(* IEC 61131-3 sources: Std_PalletMover/Class/Dana_Tm4, 1 file *)

(* ---- Dana_Tm4.st ---- *)
(*!
<Class
	Name               = "Dana_Tm4"
	Revision           = "0.0"
	RealtimeTask       = "false"
	CyclicTask         = "true"
	BackgroundTask     = "false"
	Sigmatek           = "false"
	OSInterface        = "false"
	HighPriority       = "false"
	Automatic          = "false"
	UpdateMode         = "Prescan"
	SharedCommandTable = "true"
	Objectsize         = "(900,180)">
	<Channels>
		<Server Name="ActualEncoder" Visualized="false" Initialize="false" WriteProtected="true" Retentive="false"/>
		<Server Name="ActualSpeed" Visualized="false" Initialize="false" WriteProtected="true" Retentive="false"/>
		<Server Name="ActualTorque" Visualized="false" Initialize="false" WriteProtected="true" Retentive="false"/>
		<Server Name="BatteryLevel" Visualized="false" Initialize="false" WriteProtected="true" Retentive="false"/>
		<Server Name="BatteryVoltage" Visualized="false" Initialize="false" WriteProtected="true" Retentive="false"/>
		<Server Name="InverterTemp" Visualized="false" Initialize="false" WriteProtected="true" Retentive="false"/>
		<Server Name="MotorControl" Visualized="false" Initialize="false" WriteProtected="true" Retentive="false"/>
		<Server Name="MotorError" Visualized="false" Initialize="false" WriteProtected="true" Retentive="false"/>
		<Server Name="MotorLoad" Visualized="false" Initialize="false" WriteProtected="true" Retentive="false"/>
		<Server Name="MotorState" Visualized="false" Initialize="false" WriteProtected="false" Retentive="false"/>
		<Server Name="MotorTemp" Visualized="false" Initialize="false" WriteProtected="true" Retentive="false"/>
		<Server Name="SetFeedForward" Visualized="false" Initialize="false" WriteProtected="true" Retentive="false"/>
		<Server Name="SetSpeed" Visualized="false" Initialize="false" WriteProtected="true" Retentive="false"/>
	</Channels>
	<Network Name="Dana_Tm4">
		<!-- List of Components in this network -->
		<Components>
			<Object
				Name       = "_base"
				Class      = "CanOpenWewoBase"
				Position   = "(218,120)"
				Visualized = "false">
				<Channels>
					<Server Name="Server0"/>
					<Client Name="cNode"/>
					<Client Name="ConfigData"/>
					<Client Name="Driver"/>
				</Channels>
			</Object>
		</Components>
		<Comments>
		</Comments>
		<!-- List of Connections in this network -->
		<Connections>
			<Connection Source="this.Server0" Destination="_base.Server0" Vertices="(946,210),(774,210),"/>
			<Connection Source="_base.cNode" Destination="this.cNode" Vertices="(218,270),(38,270),"/>
			<Connection Source="_base.Driver" Destination="this.Driver" Vertices="(218,210),(38,210),"/>
		</Connections>
		<!-- Headerfiles -->
		<Options>
		</Options>
	</Network>
</Class>
*)
#pragma using CanOpenWewoBase

Dana_Tm4 : CLASS
: CanOpenWewoBase
	TYPE
	  tControlWord : BINT  //! <Type Public="true" Name="tControlWord"/>
	  [
	    1 DriveEnable,
	    2 MainContactor,
	    3 BrakeRelease,
	    4 Output_01,
	    5 Output_02,
	    6 Output_03,
	    7 Output_04,
	    8 SafeStop,
	    9 Bit9,
	    10 Bit10,
	    11 Bit11,
	    12 Bit12,
	    13 Bit13,
	    14 Bit14,
	    15 Bit15,
	    16 Reset,
	  ];
#pragma pack(push, 1)
	  tCurrent : STRUCT
	    StructItem : SINT;
	    StructItem0 : SINT;
	  END_STRUCT;
#pragma pack(pop)
	  tStatusbyte : BSINT  //! <Type Public="true" Name="tStatusbyte"/>
	  [
	    1 PowerActive,
	    2 Fault,
	    3 TorqueMode,
	    4 ModeAnalog,
	    5 ModeCan,
	    6 ccwActive,
	    7 SafeStopActive,
	    8 ToggelBit,
	  ];
	END_TYPE
  //Servers:
	MotorState 	: SvrCh_gt_AgvMotorState;
	MotorLoad 	: SvrCh_DINT;
	ActualSpeed 	: SvrCh_DINT;
	ActualTorque 	: SvrCh_DINT;
	ActualEncoder 	: SvrCh_DINT;
	MotorError 	: SvrCh_DINT;
	BatteryLevel 	: SvrCh_DINT;
	InverterTemp 	: SvrCh_DINT;
	MotorTemp 	: SvrCh_DINT;
	BatteryVoltage 	: SvrCh_DINT;
	SetSpeed 	: SvrCh_DINT;
	SetFeedForward 	: SvrCh_DINT;
	MotorControl 	: SvrCh_gt_AgvMotorControl;
  //Clients:
  //Variables:
		MotorStatus 	: tStatusbyte;
		MotorCntr 	: tControlWord;
		Current 	: tCurrent;
		CurrendState 	: gt_AgvMotorState;
		ReqState 	: gt_AgvMotorState;
		LastToggelBit 	: DINT;
		LasttAlive 	: UDINT;
		MotorTimeOut 	: DINT;
  //Functions:

	FUNCTION VIRTUAL GLOBAL CyWork
		VAR_INPUT
			EAX 	: UDINT;
		END_VAR
		VAR_OUTPUT
			state (EAX) 	: UDINT := READY;
		END_VAR;

	FUNCTION GetdataCan;

	FUNCTION SetdataCan;

	FUNCTION GLOBAL Method;

	FUNCTION HandelStates;

	FUNCTION CheckError;

	FUNCTION VIRTUAL GLOBAL MotorState::Read
		VAR_OUTPUT
			output (EAX) 	: gt_AgvMotorState;
		END_VAR;

	FUNCTION VIRTUAL GLOBAL MotorState::Write
		VAR_INPUT
			input (EAX) 	: gt_AgvMotorState;
		END_VAR
		VAR_OUTPUT
			result (EAX) 	: gt_AgvMotorState;
		END_VAR;
  //Tables:
	FUNCTION @STD
		VAR_OUTPUT
			ret_code	: CONFSTATES;
		END_VAR;
	FUNCTION GLOBAL TAB @CT_;
END_CLASS;

FUNCTION VIRTUAL GLOBAL Dana_Tm4::CyWork
	VAR_INPUT
		EAX 	: UDINT;
	END_VAR
	VAR_OUTPUT
		state (EAX) 	: UDINT;(* := READY *)
	END_VAR

     GetdataCan();

     HandelStates();

     SetDataCan();

END_FUNCTION

FUNCTION Dana_Tm4::GetdataCan

    VAR
    	Pdata : ^CanObjStr;
    END_VAR

     Pdata := GetPDO(PdoId:=16#180);
    if Pdata <> nil then
         MotorStatus    := Pdata^.Data[1];
         MotorLoad      := Pdata^.Data[2];
         ActualTorque   := Pdata^.Data[3]$int;
         ActualSpeed    := Pdata^.Data[5]$int;
         ActualEncoder := Pdata^.Data[7]$int;
    END_IF;

    Pdata := GetPDO(PdoId:=16#280);
    if Pdata <> nil then
        MotorError      := Pdata^.Data[1]$int;
        BatteryLevel     :=Pdata^.Data[3];
        InverterTemp    :=Pdata^.Data[4];
        MotorTemp       :=Pdata^.Data[5]$int;
        BatteryVoltage  :=Pdata^.Data[7]$int;
    end_if;

END_FUNCTION

FUNCTION Dana_Tm4::SetdataCan

SendPDO(PdoId:=16#200, Bytes:=8, Value1:=MotorCntr$INT, Value2:=SetSpeed$int, Value3:=SetFeedForward$int, Value4:=Current$int);

END_FUNCTION

FUNCTION VIRTUAL GLOBAL Dana_Tm4::MotorState::Write
	VAR_INPUT
		input (EAX) 	: gt_AgvMotorState;
	END_VAR
	VAR_OUTPUT
		result (EAX) 	: gt_AgvMotorState;
	END_VAR

	MotorState := ::gt_AgvMotorState::M_St_Busy;;
    ReqState := input;
	result := ::gt_AgvMotorState::M_St_Busy;

END_FUNCTION

FUNCTION GLOBAL Dana_Tm4::Method

END_FUNCTION

FUNCTION Dana_Tm4::HandelStates

    case CurrendState of

        ::gt_AgvMotorState::M_St_Config:

        ::gt_AgvMotorState::M_St_Error:

        ::gt_AgvMotorState::M_St_Ready:
            CheckError();
            MotorState := ::gt_AgvMotorState::M_St_Ready;

        ::gt_AgvMotorState::M_St_Operational:
               CheckError();

        ::gt_AgvMotorState::M_St_Reset:
             if LastToggelBit <> MotorStatus.ToggelBit then
                CurrendState :=  ::gt_AgvMotorState::M_St_Ready;
                MotorState := ::gt_AgvMotorState::M_St_Ready;
            end_if;

    end_case;

    case ReqState of

          ::gt_AgvMotorState::M_St_Reset:
            MotorCntr.Reset := true;
            CurrendState :=  ::gt_AgvMotorState::M_St_Reset;
            ReqState := ::gt_AgvMotorState::M_St_Busy;
            LastToggelBit := MotorStatus.ToggelBit;

           ::gt_AgvMotorState::M_St_Busy:

    end_case;

END_FUNCTION

FUNCTION VIRTUAL GLOBAL Dana_Tm4::MotorState::Read
	VAR_OUTPUT
		output (EAX) 	: gt_AgvMotorState;
	END_VAR

    MotorState := CurrendState;
	output := MotorState;

END_FUNCTION

FUNCTION Dana_Tm4::CheckError
    if tAlive = LasttAlive then
        MotorTimeOut -=1;
        if MotorTimeOut <= 0 then
            ReqState :=   gt_AgvMotorState::M_St_Error;
         end_if;
    else
         MotorTimeOut := 200;
      LasttAlive :=  tAlive;
   end_if;

END_FUNCTION
